FUNCTION_BLOCK NodeCollection implements I_NodeCollection
VAR
	nodes : ARRAY [0..GraphFramework.MAX_NODES] OF I_Node;
	lastNode : INT := EMPTY;
END_VAR
VAR CONSTANT
	EMPTY : INT := -1;
END_VAR

METHOD PUBLIC Accept
VAR_INPUT
	Visitor : I_NodeVisitor;
END_VAR
VAR
	i : DINT;
END_VAR
FOR i := 0 TO Count - 1 DO
	GetByIndex(i).Accept(Visitor);
END_FOR
END_METHOD

PROPERTY PUBLIC Count : DINT
GET
Count := lastNode + 1;
END_GET
END_PROPERTY

METHOD PUBLIC DisposeAll
VAR
	i: INT;
END_VAR
FOR i := 0 TO lastNode DO
	IF IsValidNode(nodes[i]) THEN
		DisposeNode(nodes[i]);
		nodes[i] := 0;
	END_IF
END_FOR

lastNode := EMPTY;
END_METHOD

METHOD PUBLIC ExecuteInOrder
VAR
	nodeIndex: INT;
	nodeOrder, highestExecutionOrder : DINT;
END_VAR
highestExecutionOrder := GetHighestExecutionOrder();

FOR nodeOrder := 0 TO highestExecutionOrder DO
	FOR nodeIndex := 0 TO lastNode DO
		IF IsValidNode(nodes[nodeIndex]) THEN
			IF nodes[nodeIndex].Order = nodeOrder AND nodes[nodeIndex].mode = 0 THEN
				nodes[nodeIndex].Execute();
			END_IF
		END_IF
	END_FOR
END_FOR
END_METHOD

METHOD PUBLIC GetById : I_Node
VAR_INPUT
	Id : NodeId;
END_VAR
VAR
	i : INT;
END_VAR
FOR i := 0 TO lastNode DO
	IF  nodes[i].Id = Id THEN
		GetById := nodes[i];
		RETURN;
	END_IF
END_FOR
END_METHOD

METHOD PUBLIC GetByIndex : I_Node
VAR_INPUT
	Id : NodeId;
END_VAR
GetByIndex := nodes[Id];
END_METHOD

METHOD PUBLIC GetFirst : I_Node
IF Count = 0 THEN
	RETURN;
END_IF

GetFirst := nodes[0];
END_METHOD

METHOD PUBLIC GetHighestExecutionOrder : DINT
VAR_INPUT
END_VAR
VAR
	i : INT;
	currentOrder : DINT;
	currentHighestOrder : DINT;
END_VAR
FOR i := 0 TO lastNode DO
	currentOrder := nodes[i].Order;
	IF  currentHighestOrder <= currentOrder THEN
		currentHighestOrder := currentOrder;
	END_IF
END_FOR

GetHighestExecutionOrder := currentHighestOrder;
END_METHOD

METHOD PUBLIC GetNext : I_Node
VAR_INPUT
	CurrentNode : I_Node;
END_VAR
VAR
	i : INT;
END_VAR
IF Count = 0 THEN
	RETURN;
END_IF

IF CurrentNode = 0 THEN
	GetNext := GetFirst();
	RETURN;
END_IF

IF CurrentNode = nodes[lastNode] THEN
	GetNext := 0;
	RETURN;
END_IF

FOR i := 0 TO lastNode DO
	IF nodes[i] = CurrentNode THEN
		GetNext := nodes[i+1];
		RETURN;
	END_IF
END_FOR
END_METHOD

METHOD PUBLIC Insert : NodeId
VAR_INPUT
	node : I_Node;
END_VAR
VAR
	i : INT;
END_VAR
FOR i := 0 TO lastNode DO
	IF  nodes[i].Id = Node.Id THEN
		RETURN;
	END_IF
END_FOR

lastNode := lastNode + 1;
nodes[lastNode] := node;
END_METHOD

END_FUNCTION_BLOCK

(* stored: Version 1.1.0.1, ProductVersion 3.1.4024.12
   POU NodeCollection: Id {2c2750c5-dc73-0222-3bfb-b64d4987284f}, SpecialFunc None
   Method Accept: Id {a717681c-b528-0946-1e6e-7618985902f1}
   Property Count: Id {e9835c2c-d1ee-0ee0-2220-6784858c386a}
   Get Get: Id {fbc8e8ca-fc08-02fc-26f2-93c9b81daaab}
   Method DisposeAll: Id {a835f120-b18a-0c68-1080-8fadbc348f30}
   Method ExecuteInOrder: Id {78826cc5-34e4-0e24-0319-01868f6c2315}
   Method GetById: Id {a50f1dc9-43ab-0243-0c04-834a82271a2c}
   Method GetByIndex: Id {edf28911-bf94-050c-308d-ce5d03e562b6}
   Method GetFirst: Id {7552a64b-06ba-0c4a-1c5d-046ca697be56}
   Method GetHighestExecutionOrder: Id {25b59e23-8463-0f08-2926-2f4756fe9744}
   Method GetNext: Id {39a571bf-388e-0acb-3bb9-f334f70e7bf7}
   Method Insert: Id {2a819fd0-789a-0131-38dd-4dd9a5e26e27} *)
